PROGRAM LineChart
VAR
	TestData	: ARRAY[0..1,1..10000] OF st_Data;
	i : INT;
	Test : BOOL;
END_VAR

FOR i := 1 TO 10000 DO
	IF Test THEN
		TestData[0,i].x := i;
		TestData[0,i].y := i;
	ELSE
		TestData[0,i].x := i;
		TestData[0,i].y := 4;			
	END_IF
END_FOR

END_PROGRAM

(* stored: Version 1.1.0.1
   POU LineChart: Id {ff880aae-28d7-445f-b1dd-cc1a44a18b99}, SpecialFunc None *)
